Staubli VAL3: saveIt.pgx

program saveIt(bool& x_bSave[])
  local string l_sMessage
  local num l_nResult
  local string l_sResult
begin
end
